PROGRAM MAIN
VAR
END_VAR

END_PROGRAM

(* stored: Version 1.1.0.1
   POU MAIN: Id {1f078a04-f04d-43cc-9347-b999597687eb} *)
